FUNCTION_BLOCK TOGGLE
VAR_INPUT
	IN : BOOL;
	RESET : BOOL;
END_VAR
VAR_OUTPUT
	Q : BOOL;
END_VAR
VAR
	edge : BOOL;
END_VAR

(* This function block toggle the state of the output (Q) when the input (IN)
	transitions from a FALSE to TRUE.
	If the reset input (RESET) is true, then the output is always false *)
IF RESET THEN
	Q:=0;
ELSIF IN AND NOT edge THEN
	Q:=NOT Q;
END_IF;
edge:=IN;

END_FUNCTION_BLOCK

(* stored: Version 1.1.0.1, ProductVersion 3.1.4024.15
   POU TOGGLE: Id {df950bd4-4220-41ab-8fac-7cc6b1da6524}, SpecialFunc None *)
